// String builder function
FUNCTION F_StringBuilder : REFERENCE TO FB_StringBuilder
VAR_STAT
	fbStringBuilder : FB_StringBuilder;
END_VAR

fbStringBuilder.Clear();
F_StringBuilder REF= fbStringBuilder;

END_FUNCTION

(* stored: Version 1.1.0.1, ProductVersion 3.1.4024.4
   POU F_StringBuilder: Id {55e881ac-c530-44b9-b16a-c0ea1631cee2}, SpecialFunc None *)
